FUNCTION_BLOCK FB_Valve
VAR_INPUT
END_VAR
VAR_OUTPUT
	bDigiOut1 AT %Q* : BOOL;
	bDigiOut2 AT %Q* : BOOL;	//Für Ventile mit 2 Spulen und Mittelstellung
END_VAR
VAR
	
END_VAR

METHOD M_On
VAR_INPUT
	nChannel	: USINT;	//1 oder 2 bei Ventil mit 2 Spulen und Mittelstellung
END_VAR
IF nChannel = 1 THEN
	bDigiOut1 := TRUE;
	bDigiOut2 := FALSE;	
ELSIF nChannel = 2 THEN
	bDigiOut1 := FALSE;
	bDigiOut2 := TRUE;
ELSE
	bDigiOut1 := FALSE;
	bDigiOut2 := FALSE;
END_IF
END_METHOD

METHOD M_Off
VAR_INPUT
END_VAR
bDigiOut1 := FALSE;
bDigiOut2 := FALSE;
END_METHOD

END_FUNCTION_BLOCK

(* stored: Version 1.1.0.1, ProductVersion 3.1.0.25
   POU FB_Valve: Id {023069b1-e3a2-43dd-a646-5ec356221c42}
   Method M_On: Id {6bb4e1a2-8675-40ca-a1ba-62add57592fe}
   Method M_Off: Id {c308813f-c942-41a5-8897-3fde347bedd5} *)
